PROGRAM prgMathTesting
VAR
	noise:FB_CTRL_NOISE_GENERATOR;
	mode: E_CTRL_MODE := E_CTRL_MODE.eCTRL_MODE_ACTIVE;
	paramNoise: ST_CTRL_NOISE_GENERATOR_PARAMS := (tCtrlCycleTime := TIME#10MS, tTaskCycleTime := TIME#10MS, fAmplitude := 5);
	integrator:FB_TimeBasedIntegrator;
	addNegative: BOOL;
END_VAR

noise(
	fManSyncValue:= , 
	eMode:= mode, 
	fOut=> , 
	eState=> , 
	eErrorId=> , 
	bError=> , 
	stParams:= paramNoise);

integrator(
	tBaseTime:= T#1S, 
	rIn:= noise.fOut, 
	addNegativeValues:= addNegative, 
	bErr=> , 
	rAccumulator:= GVL_math.rIntegratorResult);

END_PROGRAM

(* stored: Version 1.1.0.1, ProductVersion 3.1.4024.12
   POU prgMathTesting: Id {d9888b1e-75bb-4e7f-97be-34b919d569a6}, SpecialFunc None *)
